TYPE FunctionResult_Log :
(
	ERROR := -1,
	BUSY := 0,
	DONE
);
END_TYPE

(* stored: Version 1.1.0.1, ProductVersion 3.1.4018.2
   DUT FunctionResult_Log: Id {ed2396a8-f253-48fa-97ec-398515224d96} *)
